FUNCTION F_Multiply : DINT
VAR_INPUT
	nNum1 : INT;
	nNum2 : INT;
END_VAR
VAR
END_VAR

F_Multiply := nNum1 * nNum2;

END_FUNCTION

(* stored: Version 1.1.0.1, ProductVersion 3.1.4024.16
   POU F_Multiply: Id {db3107e0-a955-4414-a2d0-8c4a05246579}, SpecialFunc None *)
